// TIA Portal V19 export
TYPE "C501_STU_PPP_TYPIC"
   STRUCT
      CMD { ExternalAccessible := 'False'; ExternalVisible := 'False'; ExternalWritable := 'False'} : USInt;   // Sturing pomp
      CMD_SNE { ExternalAccessible := 'False'; ExternalVisible := 'False'; ExternalWritable := 'False'} : Real;   // Sturing snelheid pomp
   END_STRUCT;
END_TYPE
